Yaskawa INFORM job: yellow_cover_planes_program.JBI

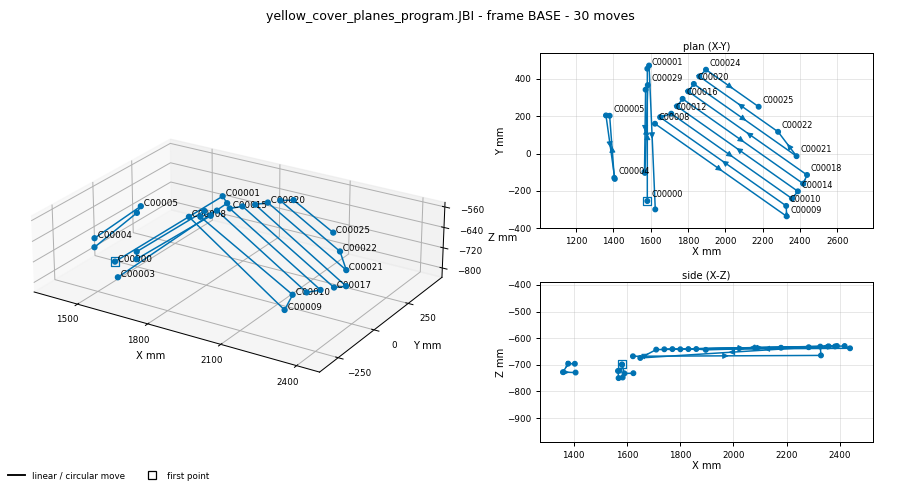
[picture p0: tool path of yellow_cover_planes_program.JBI in frame BASE, 30 of 35 moves have a stored position in this frame; points joined in program order, loops and branches not executed]
/JOB
//NAME yellow_cover_planes_program
//POS
///NPOS 30,0,30,0,0,0
///TOOL 0
///POSTYPE BASE
///RECTAN
///RCONF 0,0,0,0,0,0,0,0,0,0,0,0,0,0,0,0,0,0,0,0,0,0,0,0
C00000=1581.557084,-254.465695,-698.658352,175.000000,-89.379980,-5.000000
C00001=1581.641461,455.135296,-699.830421,175.000000,-89.379980,-5.000000
C00002=1590.973005,472.114998,-732.470039,175.000000,-89.379980,-5.000000
C00003=1624.325458,-299.337662,-731.557745,180.000000,-60.000000,0.000000
C00004=1404.542055,-129.971690,-696.082808,175.000000,-87.907858,-5.000000
C00005=1379.651191,202.851102,-695.513485,175.000000,-87.907858,-5.000000
C00006=1359.927533,204.569102,-727.628764,175.000000,-87.907858,-5.000000
C00007=1407.357819,-135.824106,-729.013741,180.000000,-60.000000,0.000000
C00008=1622.685829,160.124451,-667.902650,-175.000000,-5.000000,-5.000000
C00009=2328.760999,-336.536629,-664.734601,-175.000000,-5.000000,-5.000000
C00010=2326.133960,-280.514676,-631.610601,-175.000000,-5.000000,-5.000000
C00011=1650.217102,194.932714,-674.231601,-175.000000,-5.000000,-5.000000
C00012=1710.081050,213.954495,-642.913601,-175.000000,-5.000000,-5.000000
C00013=2357.649652,-241.552419,-630.623601,-175.000000,-5.000000,-5.000000
C00014=2388.821817,-202.348521,-629.445601,-175.000000,-5.000000,-5.000000
C00015=1740.541625,253.658932,-641.712601,-175.000000,-5.000000,-5.000000
C00016=1770.860701,293.462903,-641.070601,-175.000000,-5.000000,-5.000000
C00017=2417.595026,-161.457171,-629.496601,-175.000000,-5.000000,-5.000000
C00018=2437.879871,-114.595011,-637.997601,-175.000000,-5.000000,-5.000000
C00019=1800.690661,333.610922,-641.662601,-175.000000,-5.000000,-5.000000
C00020=1830.930399,373.470700,-640.952601,-175.000000,-5.000000,-5.000000
C00021=2381.704006,-13.949544,-630.943601,-175.000000,-5.000000,-5.000000
C00022=2282.748521,116.787582,-633.974601,-175.000000,-5.000000,-5.000000
C00023=1860.562423,413.757950,-640.681601,-175.000000,-5.000000,-5.000000
C00024=1896.211482,449.818864,-643.827601,-175.000000,-5.000000,-5.000000
C00025=2178.697905,251.114792,-635.895601,-175.000000,-5.000000,-5.000000
C00026=1572.425096,342.716431,-721.791802,-5.000000,-83.940775,175.000000
C00027=1566.552181,-97.925944,-723.094401,-5.000000,-83.940775,175.000000
C00028=1568.787698,-103.595995,-749.985053,-5.000000,-83.940775,175.000000
C00029=1584.096577,367.141073,-747.634441,180.000000,-60.000000,0.000000
///POSTYPE PULSE
///PULSE
EC00000=17408.0
EC00001=17408.0
EC00002=17408.0
EC00003=17408.0
EC00004=95232.0
EC00005=95232.0
EC00006=95232.0
EC00007=95232.0
EC00008=240640.0
EC00009=240640.0
EC00010=240640.0
EC00011=240640.0
EC00012=240640.0
EC00013=240640.0
EC00014=240640.0
EC00015=240640.0
EC00016=240640.0
EC00017=240640.0
EC00018=240640.0
EC00019=240640.0
EC00020=240640.0
EC00021=240640.0
EC00022=240640.0
EC00023=240640.0
EC00024=240640.0
EC00025=240640.0
EC00026=278528.0
EC00027=278528.0
EC00028=278528.0
EC00029=278528.0
//INST
///DATE 2023/08/16 14:03
///ATTR SC,RW,RJ
////FRAME BASE
///GROUP1 RB1,ST1
NOP
MOVJ P009 EX000 VJ=15.00
MOVJ C00000 EC00000 VJ=15.0
CALL JOB:SPYON
MOVL C00001 EC00001 V=150.0
MOVL C00002 EC00002 V=150.0
MOVL C00003 EC00003 V=150.0
CALL JOB:SPYOF
MOVJ P009 VJ=15.00
MOVJ C00004 EC00004 VJ=15.0
CALL JOB:SPYON
MOVL C00005 EC00005 V=150.0
MOVL C00006 EC00006 V=150.0
MOVL C00007 EC00007 V=150.0
CALL JOB:SPYOF
MOVJ P009 VJ=15.00
MOVJ C00008 EC00008 VJ=15.0
CALL JOB:SPYON
MOVL C00009 EC00009 V=150.0
MOVL C00010 EC00010 V=150.0
MOVL C00011 EC00011 V=150.0
MOVL C00012 EC00012 V=150.0
MOVL C00013 EC00013 V=150.0
MOVL C00014 EC00014 V=150.0
MOVL C00015 EC00015 V=150.0
MOVL C00016 EC00016 V=150.0
MOVL C00017 EC00017 V=150.0
MOVL C00018 EC00018 V=150.0
MOVL C00019 EC00019 V=150.0
MOVL C00020 EC00020 V=150.0
MOVL C00021 EC00021 V=150.0
MOVL C00022 EC00022 V=150.0
MOVL C00023 EC00023 V=150.0
MOVL C00024 EC00024 V=150.0
MOVL C00025 EC00025 V=150.0
CALL JOB:SPYOF
MOVJ P009 VJ=15.00
MOVJ C00026 EC00026 VJ=15.0
CALL JOB:SPYON
MOVL C00027 EC00027 V=150.0
MOVL C00028 EC00028 V=150.0
MOVL C00029 EC00029 V=150.0
CALL JOB:SPYOF
MOVJ P009 VJ=15.00
END
